   AIO_8B0E.RAW_NAME := 'Thermal Resistance - 3-wire (Cu10 climate - 426)';
   AIO_8B0E.___________0030_1 := false;
   AIO_8B0E.___________0030_2 := false;
   AIO_8B0E.PARAM_TYPE := 16#07;
   AIO_8B0E.PARAM_RANGE := 16#0E;
   AIO_8B0E.PARAM_COEF := 16#0B;
   AIO_8B0E.VALUE_COEF := 0.00426;
   AIO_8C0E.AIO_CODE := 16#8C0E;
   AIO_8C0E.___________0020_0 := false;
   AIO_8C0E.___________0010_2 := false;
   AIO_8C0E.RAW_MIN := -5000;
   AIO_8C0E.RAW_MAX := 15000;
   AIO_8C0E.RAW_NAME := 'Thermal Resistance - 3-wire (Cu10 climate - 427)';
   AIO_8C0E.___________0030_1 := false;
   AIO_8C0E.___________0030_2 := false;
   AIO_8C0E.PARAM_TYPE := 16#07;
   AIO_8C0E.PARAM_RANGE := 16#0E;
   AIO_8C0E.PARAM_COEF := 16#0C;
   AIO_8C0E.VALUE_COEF := 0.00427;
   AIO_8D0E.AIO_CODE := 16#8D0E;
   AIO_8D0E.___________0020_0 := false;
   AIO_8D0E.___________0010_2 := false;
   AIO_8D0E.RAW_MIN := -1800;
   AIO_8D0E.RAW_MAX := 15000;
   AIO_8D0E.RAW_NAME := 'Thermal Resistance - 3-wire (Cu10 climate - 428)';
   AIO_8D0E.___________0030_1 := false;
   AIO_8D0E.___________0030_2 := false;
   AIO_8D0E.PARAM_TYPE := 16#07;
   AIO_8D0E.PARAM_RANGE := 16#0E;
   AIO_8D0E.PARAM_COEF := 16#0D;
   AIO_8D0E.VALUE_COEF := 0.00428;
   AIO_8B0F.AIO_CODE := 16#8B0F;
   AIO_8B0F.___________0020_0 := false;
   AIO_8B0F.___________0010_2 := false;
   AIO_8B0F.RAW_MIN := -500;
   AIO_8B0F.RAW_MAX := 2000;
   AIO_8B0F.RAW_NAME := 'Thermal Resistance - 3-wire (Cu10 standard - 426)';
   AIO_8B0F.___________0030_1 := false;
   AIO_8B0F.___________0030_2 := false;
   AIO_8B0F.PARAM_TYPE := 16#07;
   AIO_8B0F.PARAM_RANGE := 16#0F;
   AIO_8B0F.PARAM_COEF := 16#0B;
   AIO_8B0F.VALUE_COEF := 0.00426;
   AIO_8C0F.AIO_CODE := 16#8C0F;
   AIO_8C0F.___________0020_0 := false;
   AIO_8C0F.___________0010_2 := false;
   AIO_8C0F.RAW_MIN := -2000;
   AIO_8C0F.RAW_MAX := 2600;
   AIO_8C0F.RAW_NAME := 'Thermal Resistance - 3-wire (Cu10 standard - 427)';
   AIO_8C0F.___________0030_1 := false;
   AIO_8C0F.___________0030_2 := false;
   AIO_8C0F.PARAM_TYPE := 16#07;
   AIO_8C0F.PARAM_RANGE := 16#0F;
   AIO_8C0F.PARAM_COEF := 16#0C;
   AIO_8C0F.VALUE_COEF := 0.00427;
   AIO_8D0F.AIO_CODE := 16#8D0F;
   AIO_8D0F.___________0020_0 := false;
   AIO_8D0F.___________0010_2 := false;
   AIO_8D0F.RAW_MIN := -1800;
   AIO_8D0F.RAW_MAX := 2000;
   AIO_8D0F.RAW_NAME := 'Thermal Resistance - 3-wire (Cu10 standard - 428)';
   AIO_8D0F.___________0030_1 := false;
   AIO_8D0F.___________0030_2 := false;
   AIO_8D0F.PARAM_TYPE := 16#07;
   AIO_8D0F.PARAM_RANGE := 16#0F;
   AIO_8D0F.PARAM_COEF := 16#0D;
   AIO_8D0F.VALUE_COEF := 0.00428;
   AIO_8B19.AIO_CODE := 16#8B19;
   AIO_8B19.___________0020_0 := false;
   AIO_8B19.___________0010_2 := false;
   AIO_8B19.RAW_MIN := -5000;
   AIO_8B19.RAW_MAX := 15000;
   AIO_8B19.RAW_NAME := 'Thermal Resistance - 3-wire (Cu50 climate - 426)';
   AIO_8B19.___________0030_1 := false;
   AIO_8B19.___________0030_2 := false;
   AIO_8B19.PARAM_TYPE := 16#07;
   AIO_8B19.PARAM_RANGE := 16#19;
   AIO_8B19.PARAM_COEF := 16#0B;
   AIO_8B19.VALUE_COEF := 0.00426;
   AIO_8C19.AIO_CODE := 16#8C19;
   AIO_8C19.___________0020_0 := false;
   AIO_8C19.___________0010_2 := false;
   AIO_8C19.RAW_MIN := -5000;
   AIO_8C19.RAW_MAX := 15000;
   AIO_8C19.RAW_NAME := 'Thermal Resistance - 3-wire (Cu50 climate - 427)';
   AIO_8C19.___________0030_1 := false;
   AIO_8C19.___________0030_2 := false;
   AIO_8C19.PARAM_TYPE := 16#07;
   AIO_8C19.PARAM_RANGE := 16#19;
   AIO_8C19.PARAM_COEF := 16#0C;
   AIO_8C19.VALUE_COEF := 0.00427;
   AIO_8D19.AIO_CODE := 16#8D19;
   AIO_8D19.___________0020_0 := false;
   AIO_8D19.___________0010_2 := false;
   AIO_8D19.RAW_MIN := -5000;
   AIO_8D19.RAW_MAX := 15000;
   AIO_8D19.RAW_NAME := 'Thermal Resistance - 3-wire (Cu50 climate - 428)';
   AIO_8D19.___________0030_1 := false;
   AIO_8D19.___________0030_2 := false;
   AIO_8D19.PARAM_TYPE := 16#07;
   AIO_8D19.PARAM_RANGE := 16#19;
   AIO_8D19.PARAM_COEF := 16#0D;
   AIO_8D19.VALUE_COEF := 0.00428;
   AIO_8B18.AIO_CODE := 16#8B18;
   AIO_8B18.___________0020_0 := false;
   AIO_8B18.___________0010_2 := false;
   AIO_8B18.RAW_MIN := -500;
   AIO_8B18.RAW_MAX := 2000;
   AIO_8B18.RAW_NAME := 'Thermal Resistance - 3-wire (Cu50 standard - 426)';
   AIO_8B18.___________0030_1 := false;
   AIO_8B18.___________0030_2 := false;
   AIO_8B18.PARAM_TYPE := 16#07;
   AIO_8B18.PARAM_RANGE := 16#18;
   AIO_8B18.PARAM_COEF := 16#0B;
   AIO_8B18.VALUE_COEF := 0.00426;
   AIO_8C18.AIO_CODE := 16#8C18;
   AIO_8C18.___________0020_0 := false;
   AIO_8C18.___________0010_2 := false;
   AIO_8C18.RAW_MIN := -2000;
   AIO_8C18.RAW_MAX := 2600;
   AIO_8C18.RAW_NAME := 'Thermal Resistance - 3-wire (Cu50 standard - 427)';
   AIO_8C18.___________0030_1 := false;
   AIO_8C18.___________0030_2 := false;
   AIO_8C18.PARAM_TYPE := 16#07;
   AIO_8C18.PARAM_RANGE := 16#18;
   AIO_8C18.PARAM_COEF := 16#0C;
   AIO_8C18.VALUE_COEF := 0.00427;
   AIO_8D18.AIO_CODE := 16#8D18;
   AIO_8D18.___________0020_0 := false;
   AIO_8D18.___________0010_2 := false;
   AIO_8D18.RAW_MIN := -1800;
   AIO_8D18.RAW_MAX := 2000;
   AIO_8D18.RAW_NAME := 'Thermal Resistance - 3-wire (Cu50 standard - 428)';
   AIO_8D18.___________0030_1 := false;
   AIO_8D18.___________0030_2 := false;
   AIO_8D18.PARAM_TYPE := 16#07;
   AIO_8D18.PARAM_RANGE := 16#18;
   AIO_8D18.PARAM_COEF := 16#0D;
   AIO_8D18.VALUE_COEF := 0.00428;
   AIO_8B1B.AIO_CODE := 16#8B1B;
   AIO_8B1B.___________0020_0 := false;
   AIO_8B1B.___________0010_2 := false;
   AIO_8B1B.RAW_MIN := -5000;
   AIO_8B1B.RAW_MAX := 15000;
   AIO_8B1B.RAW_NAME := 'Thermal Resistance - 3-wire (Cu100 climate - 426)';
   AIO_8B1B.___________0030_1 := false;
   AIO_8B1B.___________0030_2 := false;
   AIO_8B1B.PARAM_TYPE := 16#07;
   AIO_8B1B.PARAM_RANGE := 16#1B;
   AIO_8B1B.PARAM_COEF := 16#0B;
   AIO_8B1B.VALUE_COEF := 0.00426;
   AIO_8C1B.AIO_CODE := 16#8C1B;
   AIO_8C1B.___________0020_0 := false;
   AIO_8C1B.___________0010_2 := false;
   AIO_8C1B.RAW_MIN := -5000;
   AIO_8C1B.RAW_MAX := 15000;
   AIO_8C1B.RAW_NAME := 'Thermal Resistance - 3-wire (Cu100 climate - 427)';
   AIO_8C1B.___________0030_1 := false;
   AIO_8C1B.___________0030_2 := false;
   AIO_8C1B.PARAM_TYPE := 16#07;
   AIO_8C1B.PARAM_RANGE := 16#1B;
   AIO_8C1B.PARAM_COEF := 16#0C;
   AIO_8C1B.VALUE_COEF := 0.00427;
   AIO_8D1B.AIO_CODE := 16#8D1B;
   AIO_8D1B.___________0020_0 := false;
   AIO_8D1B.___________0010_2 := false;
   AIO_8D1B.RAW_MIN := -5000;
   AIO_8D1B.RAW_MAX := 15000;
   AIO_8D1B.RAW_NAME := 'Thermal Resistance - 3-wire (Cu100 climate - 428)';
   AIO_8D1B.___________0030_1 := false;
   AIO_8D1B.___________0030_2 := false;
   AIO_8D1B.PARAM_TYPE := 16#07;
   AIO_8D1B.PARAM_RANGE := 16#1B;
   AIO_8D1B.PARAM_COEF := 16#0D;
   AIO_8D1B.VALUE_COEF := 0.00428;
   AIO_8B1A.AIO_CODE := 16#8B1A;
   AIO_8B1A.___________0020_0 := false;
   AIO_8B1A.___________0010_2 := false;
   AIO_8B1A.RAW_MIN := -500;
   AIO_8B1A.RAW_MAX := 2000;
   AIO_8B1A.RAW_NAME := 'Thermal Resistance - 3-wire (Cu100 standard - 426)';
   AIO_8B1A.___________0030_1 := false;
   AIO_8B1A.___________0030_2 := false;
   AIO_8B1A.PARAM_TYPE := 16#07;
   AIO_8B1A.PARAM_RANGE := 16#1A;
   AIO_8B1A.PARAM_COEF := 16#0B;
   AIO_8B1A.VALUE_COEF := 0.00426;
   AIO_8C1A.AIO_CODE := 16#8C1A;
   AIO_8C1A.___________0020_0 := false;
   AIO_8C1A.___________0010_2 := false;
   AIO_8C1A.RAW_MIN := -2000;
   AIO_8C1A.RAW_MAX := 2600;
   AIO_8C1A.RAW_NAME := 'Thermal Resistance - 3-wire (Cu100 standard - 427)';
   AIO_8C1A.___________0030_1 := false;
   AIO_8C1A.___________0030_2 := false;
   AIO_8C1A.PARAM_TYPE := 16#07;
   AIO_8C1A.PARAM_RANGE := 16#1A;
   AIO_8C1A.PARAM_COEF := 16#0C;
   AIO_8C1A.VALUE_COEF := 0.00427;
   AIO_8D1A.AIO_CODE := 16#8D1A;
   AIO_8D1A.___________0020_0 := false;
   AIO_8D1A.___________0010_2 := false;
   AIO_8D1A.RAW_MIN := -1800;
   AIO_8D1A.RAW_MAX := 2000;
   AIO_8D1A.RAW_NAME := 'Thermal Resistance - 3-wire (Cu100 standard - 428)';
   AIO_8D1A.___________0030_1 := false;
   AIO_8D1A.___________0030_2 := false;
   AIO_8D1A.PARAM_TYPE := 16#07;
   AIO_8D1A.PARAM_RANGE := 16#1A;
   AIO_8D1A.PARAM_COEF := 16#0D;
   AIO_8D1A.VALUE_COEF := 0.00428;
   AIO_8A1D.AIO_CODE := 16#8A1D;
   AIO_8A1D.___________0020_0 := false;
   AIO_8A1D.___________0010_2 := false;
   AIO_8A1D.RAW_MIN := -6000;
   AIO_8A1D.RAW_MAX := 13000;
   AIO_8A1D.RAW_NAME := 'Thermal Resistance - 3-wire (LG-Ni1000 climate - 500)';
   AIO_8A1D.___________0030_1 := false;
   AIO_8A1D.___________0030_2 := false;
   AIO_8A1D.PARAM_TYPE := 16#07;
   AIO_8A1D.PARAM_RANGE := 16#1D;
   AIO_8A1D.PARAM_COEF := 16#0A;
   AIO_8A1D.VALUE_COEF := 0.005;
   AIO_8A1C.AIO_CODE := 16#8A1C;
   AIO_8A1C.___________0020_0 := false;
   AIO_8A1C.___________0010_2 := false;
   AIO_8A1C.RAW_MIN := -600;
   AIO_8A1C.RAW_MAX := 2500;
   AIO_8A1C.RAW_NAME := 'Thermal Resistance - 3-wire (LG-Ni1000 standard - 500)';
   AIO_8A1C.___________0030_1 := false;
   AIO_8A1C.___________0030_2 := false;
   AIO_8A1C.PARAM_TYPE := 16#07;
   AIO_8A1C.PARAM_RANGE := 16#1C;
   AIO_8A1C.PARAM_COEF := 16#0A;
   AIO_8A1C.VALUE_COEF := 0.005;
   AIO_871F.AIO_CODE := 16#871F;
   AIO_871F.___________0020_0 := false;
   AIO_871F.___________0010_2 := false;
   AIO_871F.RAW_MIN := -6000;
   AIO_871F.RAW_MAX := 13000;
   AIO_871F.RAW_NAME := 'Thermal Resistance - 3-wire (Ni10 climate - 617)';
   AIO_871F.___________0030_1 := false;
   AIO_871F.___________0030_2 := false;
   AIO_871F.PARAM_TYPE := 16#07;
   AIO_871F.PARAM_RANGE := 16#1F;
   AIO_871F.PARAM_COEF := 16#07;
   AIO_871F.VALUE_COEF := 0.00617;
   AIO_881F.AIO_CODE := 16#881F;
   AIO_881F.___________0020_0 := false;
   AIO_881F.___________0010_2 := false;
   AIO_881F.RAW_MIN := -6000;
   AIO_881F.RAW_MAX := 13000;
   AIO_881F.RAW_NAME := 'Thermal Resistance - 3-wire (Ni10 climate - 618)';
   AIO_881F.___________0030_1 := false;
   AIO_881F.___________0030_2 := false;
   AIO_881F.PARAM_TYPE := 16#07;
   AIO_881F.PARAM_RANGE := 16#1F;
   AIO_881F.PARAM_COEF := 16#08;
   AIO_881F.VALUE_COEF := 0.00618;
   AIO_891F.AIO_CODE := 16#891F;
   AIO_891F.___________0020_0 := false;
   AIO_891F.___________0010_2 := false;
   AIO_891F.RAW_MIN := -6000;
   AIO_891F.RAW_MAX := 13000;
   AIO_891F.RAW_NAME := 'Thermal Resistance - 3-wire (Ni10 climate - 672)';
   AIO_891F.___________0030_1 := false;
   AIO_891F.___________0030_2 := false;
   AIO_891F.PARAM_TYPE := 16#07;
   AIO_891F.PARAM_RANGE := 16#1F;
   AIO_891F.PARAM_COEF := 16#09;
   AIO_891F.VALUE_COEF := 0.00672;
   AIO_871E.AIO_CODE := 16#871E;
   AIO_871E.___________0020_0 := false;
   AIO_871E.___________0010_2 := false;
   AIO_871E.RAW_MIN := -600;
   AIO_871E.RAW_MAX := 1800;
   AIO_871E.RAW_NAME := 'Thermal Resistance - 3-wire (Ni10 standard - 617)';
   AIO_871E.___________0030_1 := false;
   AIO_871E.___________0030_2 := false;
   AIO_871E.PARAM_TYPE := 16#07;
   AIO_871E.PARAM_RANGE := 16#1E;
   AIO_871E.PARAM_COEF := 16#07;
   AIO_871E.VALUE_COEF := 0.00617;
   AIO_881E.AIO_CODE := 16#881E;
   AIO_881E.___________0020_0 := false;
   AIO_881E.___________0010_2 := false;
   AIO_881E.RAW_MIN := -600;
   AIO_881E.RAW_MAX := 2500;
   AIO_881E.RAW_NAME := 'Thermal Resistance - 3-wire (Ni10 standard - 618)';
   AIO_881E.___________0030_1 := false;
   AIO_881E.___________0030_2 := false;
   AIO_881E.PARAM_TYPE := 16#07;
   AIO_881E.PARAM_RANGE := 16#1E;
   AIO_881E.PARAM_COEF := 16#08;
   AIO_881E.VALUE_COEF := 0.00618;
   AIO_891E.AIO_CODE := 16#891E;
   AIO_891E.___________0020_0 := false;
   AIO_891E.___________0010_2 := false;
   AIO_891E.RAW_MIN := -600;
   AIO_891E.RAW_MAX := 2500;
   AIO_891E.RAW_NAME := 'Thermal Resistance - 3-wire (Ni10 standard - 672)';
   AIO_891E.___________0030_1 := false;
   AIO_891E.___________0030_2 := false;
   AIO_891E.PARAM_TYPE := 16#07;
   AIO_891E.PARAM_RANGE := 16#1E;
   AIO_891E.PARAM_COEF := 16#09;
   AIO_891E.VALUE_COEF := 0.00672;
   AIO_870D.AIO_CODE := 16#870D;
   AIO_870D.___________0020_0 := false;
   AIO_870D.___________0010_2 := false;
   AIO_870D.RAW_MIN := -6000;
   AIO_870D.RAW_MAX := 13000;
   AIO_870D.RAW_NAME := 'Thermal Resistance - 3-wire (Ni120 climate - 617)';
   AIO_870D.___________0030_1 := false;
   AIO_870D.___________0030_2 := false;
   AIO_870D.PARAM_TYPE := 16#07;
   AIO_870D.PARAM_RANGE := 16#0D;
   AIO_870D.PARAM_COEF := 16#07;
   AIO_870D.VALUE_COEF := 0.00617;
   AIO_880D.AIO_CODE := 16#880D;
   AIO_880D.___________0020_0 := false;
   AIO_880D.___________0010_2 := false;
   AIO_880D.RAW_MIN := -6000;
   AIO_880D.RAW_MAX := 13000;
   AIO_880D.RAW_NAME := 'Thermal Resistance - 3-wire (Ni120 climate - 618)';
   AIO_880D.___________0030_1 := false;
   AIO_880D.___________0030_2 := false;
   AIO_880D.PARAM_TYPE := 16#07;
   AIO_880D.PARAM_RANGE := 16#0D;
   AIO_880D.PARAM_COEF := 16#08;
   AIO_880D.VALUE_COEF := 0.00618;
   AIO_890D.AIO_CODE := 16#890D;
   AIO_890D.___________0020_0 := false;
   AIO_890D.___________0010_2 := false;
   AIO_890D.RAW_MIN := -6000;
   AIO_890D.RAW_MAX := 13000;
   AIO_890D.RAW_NAME := 'Thermal Resistance - 3-wire (Ni120 climate - 672)';
   AIO_890D.___________0030_1 := false;
   AIO_890D.___________0030_2 := false;
   AIO_890D.PARAM_TYPE := 16#07;
   AIO_890D.PARAM_RANGE := 16#0D;
   AIO_890D.PARAM_COEF := 16#09;
   AIO_890D.VALUE_COEF := 0.00672;
   AIO_870C.AIO_CODE := 16#870C;
   AIO_870C.___________0020_0 := false;
   AIO_870C.___________0010_2 := false;
   AIO_870C.RAW_MIN := -600;
   AIO_870C.RAW_MAX := 1800;
   AIO_870C.RAW_NAME := 'Thermal Resistance - 3-wire (Ni120 standard - 617)';
   AIO_870C.___________0030_1 := false;
   AIO_870C.___________0030_2 := false;
   AIO_870C.PARAM_TYPE := 16#07;
   AIO_870C.PARAM_RANGE := 16#0C;
   AIO_870C.PARAM_COEF := 16#07;
   AIO_870C.VALUE_COEF := 0.00617;
   AIO_880C.AIO_CODE := 16#880C;
   AIO_880C.___________0020_0 := false;
   AIO_880C.___________0010_2 := false;
   AIO_880C.RAW_MIN := -600;
   AIO_880C.RAW_MAX := 2500;
   AIO_880C.RAW_NAME := 'Thermal Resistance - 3-wire (Ni120 standard - 618)';
   AIO_880C.___________0030_1 := false;
   AIO_880C.___________0030_2 := false;
   AIO_880C.PARAM_TYPE := 16#07;
   AIO_880C.PARAM_RANGE := 16#0C;
   AIO_880C.PARAM_COEF := 16#08;
   AIO_880C.VALUE_COEF := 0.00618;
   AIO_890C.AIO_CODE := 16#890C;
   AIO_890C.___________0020_0 := false;
   AIO_890C.___________0010_2 := false;
   AIO_890C.RAW_MIN := -600;
   AIO_890C.RAW_MAX := 2500;
   AIO_890C.RAW_NAME := 'Thermal Resistance - 3-wire (Ni120 standard - 672)';
   AIO_890C.___________0030_1 := false;
   AIO_890C.___________0030_2 := false;
   AIO_890C.PARAM_TYPE := 16#07;
   AIO_890C.PARAM_RANGE := 16#0C;
   AIO_890C.PARAM_COEF := 16#09;
   AIO_890C.VALUE_COEF := 0.00672;
   AIO_8701.AIO_CODE := 16#8701;
   AIO_8701.___________0020_0 := false;
   AIO_8701.___________0010_2 := false;
   AIO_8701.RAW_MIN := -6000;
   AIO_8701.RAW_MAX := 13000;
   AIO_8701.RAW_NAME := 'Thermal Resistance - 3-wire (Ni100 climate - 617)';
   AIO_8701.___________0030_1 := false;
   AIO_8701.___________0030_2 := false;
   AIO_8701.PARAM_TYPE := 16#07;
   AIO_8701.PARAM_RANGE := 16#01;
   AIO_8701.PARAM_COEF := 16#07;
   AIO_8701.VALUE_COEF := 0.00617;
   AIO_8801.AIO_CODE := 16#8801;
   AIO_8801.___________0020_0 := false;
   AIO_8801.___________0010_2 := false;
   AIO_8801.RAW_MIN := -6000;
   AIO_8801.RAW_MAX := 13000;
   AIO_8801.RAW_NAME := 'Thermal Resistance - 3-wire (Ni100 climate - 618)';
   AIO_8801.___________0030_1 := false;
   AIO_8801.___________0030_2 := false;
   AIO_8801.PARAM_TYPE := 16#07;
   AIO_8801.PARAM_RANGE := 16#01;
   AIO_8801.PARAM_COEF := 16#08;
   AIO_8801.VALUE_COEF := 0.00618;
   AIO_8901.AIO_CODE := 16#8901;
   AIO_8901.___________0020_0 := false;
   AIO_8901.___________0010_2 := false;
   AIO_8901.RAW_MIN := -6000;
   AIO_8901.RAW_MAX := 13000;
   AIO_8901.RAW_NAME := 'Thermal Resistance - 3-wire (Ni100 climate - 672)';
   AIO_8901.___________0030_1 := false;
   AIO_8901.___________0030_2 := false;
   AIO_8901.PARAM_TYPE := 16#07;
   AIO_8901.PARAM_RANGE := 16#01;
   AIO_8901.PARAM_COEF := 16#09;
   AIO_8901.VALUE_COEF := 0.00672;
   AIO_8703.AIO_CODE := 16#8703;
   AIO_8703.___________0020_0 := false;
   AIO_8703.___________0010_2 := false;
   AIO_8703.RAW_MIN := -600;
   AIO_8703.RAW_MAX := 1800;
   AIO_8703.RAW_NAME := 'Thermal Resistance - 3-wire (Ni100 standard - 617)';
   AIO_8703.___________0030_1 := false;
   AIO_8703.___________0030_2 := false;
   AIO_8703.PARAM_TYPE := 16#07;
   AIO_8703.PARAM_RANGE := 16#03;
   AIO_8703.PARAM_COEF := 16#07;
   AIO_8703.VALUE_COEF := 0.00617;
   AIO_8803.AIO_CODE := 16#8803;
   AIO_8803.___________0020_0 := false;
   AIO_8803.___________0010_2 := false;
   AIO_8803.RAW_MIN := -600;
   AIO_8803.RAW_MAX := 2500;
   AIO_8803.RAW_NAME := 'Thermal Resistance - 3-wire (Ni100 standard - 618)';
   AIO_8803.___________0030_1 := false;
   AIO_8803.___________0030_2 := false;
   AIO_8803.PARAM_TYPE := 16#07;
   AIO_8803.PARAM_RANGE := 16#03;
   AIO_8803.PARAM_COEF := 16#08;
   AIO_8803.VALUE_COEF := 0.00618;
   AIO_8903.AIO_CODE := 16#8903;
   AIO_8903.___________0020_0 := false;
   AIO_8903.___________0010_2 := false;
   AIO_8903.RAW_MIN := -600;
   AIO_8903.RAW_MAX := 2500;
   AIO_8903.RAW_NAME := 'Thermal Resistance - 3-wire (Ni100 standard - 672)';
   AIO_8903.___________0030_1 := false;
   AIO_8903.___________0030_2 := false;
   AIO_8903.PARAM_TYPE := 16#07;
   AIO_8903.PARAM_RANGE := 16#03;
   AIO_8903.PARAM_COEF := 16#09;
   AIO_8903.VALUE_COEF := 0.00672;
   AIO_8711.AIO_CODE := 16#8711;
   AIO_8711.___________0020_0 := false;
   AIO_8711.___________0010_2 := false;
   AIO_8711.RAW_MIN := -6000;
   AIO_8711.RAW_MAX := 13000;
   AIO_8711.RAW_NAME := 'Thermal Resistance - 3-wire (Ni200 climate - 617)';
   AIO_8711.___________0030_1 := false;
   AIO_8711.___________0030_2 := false;
   AIO_8711.PARAM_TYPE := 16#07;
   AIO_8711.PARAM_RANGE := 16#11;
   AIO_8711.PARAM_COEF := 16#07;
   AIO_8711.VALUE_COEF := 0.00617;
   AIO_8811.AIO_CODE := 16#8811;
   AIO_8811.___________0020_0 := false;
   AIO_8811.___________0010_2 := false;
   AIO_8811.RAW_MIN := -6000;
   AIO_8811.RAW_MAX := 13000;
   AIO_8811.RAW_NAME := 'Thermal Resistance - 3-wire (Ni200 climate - 618)';
   AIO_8811.___________0030_1 := false;
   AIO_8811.___________0030_2 := false;
   AIO_8811.PARAM_TYPE := 16#07;
   AIO_8811.PARAM_RANGE := 16#11;
   AIO_8811.PARAM_COEF := 16#08;
   AIO_8811.VALUE_COEF := 0.00618;
   AIO_8911.AIO_CODE := 16#8911;
   AIO_8911.___________0020_0 := false;
   AIO_8911.___________0010_2 := false;
   AIO_8911.RAW_MIN := -6000;
   AIO_8911.RAW_MAX := 13000;
   AIO_8911.RAW_NAME := 'Thermal Resistance - 3-wire (Ni200 climate - 672)';
   AIO_8911.___________0030_1 := false;
   AIO_8911.___________0030_2 := false;
   AIO_8911.PARAM_TYPE := 16#07;
   AIO_8911.PARAM_RANGE := 16#11;
   AIO_8911.PARAM_COEF := 16#09;
   AIO_8911.VALUE_COEF := 0.00672;
   AIO_8710.AIO_CODE := 16#8710;
   AIO_8710.___________0020_0 := false;
   AIO_8710.___________0010_2 := false;
   AIO_8710.RAW_MIN := -600;
   AIO_8710.RAW_MAX := 1800;
   AIO_8710.RAW_NAME := 'Thermal Resistance - 3-wire (Ni200 standard - 617)';
   AIO_8710.___________0030_1 := false;
   AIO_8710.___________0030_2 := false;
   AIO_8710.PARAM_TYPE := 16#07;
   AIO_8710.PARAM_RANGE := 16#10;
   AIO_8710.PARAM_COEF := 16#07;
   AIO_8710.VALUE_COEF := 0.00617;
   AIO_8810.AIO_CODE := 16#8810;
   AIO_8810.___________0020_0 := false;
   AIO_8810.___________0010_2 := false;
   AIO_8810.RAW_MIN := -600;
   AIO_8810.RAW_MAX := 2500;
   AIO_8810.RAW_NAME := 'Thermal Resistance - 3-wire (Ni200 standard - 618)';
   AIO_8810.___________0030_1 := false;
   AIO_8810.___________0030_2 := false;
   AIO_8810.PARAM_TYPE := 16#07;
   AIO_8810.PARAM_RANGE := 16#10;
   AIO_8810.PARAM_COEF := 16#08;
   AIO_8810.VALUE_COEF := 0.00618;
   AIO_8910.AIO_CODE := 16#8910;
   AIO_8910.___________0020_0 := false;
   AIO_8910.___________0010_2 := false;
   AIO_8910.RAW_MIN := -600;
   AIO_8910.RAW_MAX := 2500;
   AIO_8910.RAW_NAME := 'Thermal Resistance - 3-wire (Ni200 standard - 672)';
   AIO_8910.___________0030_1 := false;
   AIO_8910.___________0030_2 := false;
   AIO_8910.PARAM_TYPE := 16#07;
   AIO_8910.PARAM_RANGE := 16#10;
   AIO_8910.PARAM_COEF := 16#09;
   AIO_8910.VALUE_COEF := 0.00672;
   AIO_8713.AIO_CODE := 16#8713;
   AIO_8713.___________0020_0 := false;
   AIO_8713.___________0010_2 := false;
   AIO_8713.RAW_MIN := -6000;
   AIO_8713.RAW_MAX := 13000;
   AIO_8713.RAW_NAME := 'Thermal Resistance - 3-wire (Ni500 climate - 617)';
   AIO_8713.___________0030_1 := false;
   AIO_8713.___________0030_2 := false;
   AIO_8713.PARAM_TYPE := 16#07;
   AIO_8713.PARAM_RANGE := 16#13;
   AIO_8713.PARAM_COEF := 16#07;
   AIO_8713.VALUE_COEF := 0.00617;
   AIO_8813.AIO_CODE := 16#8813;
   AIO_8813.___________0020_0 := false;
   AIO_8813.___________0010_2 := false;
   AIO_8813.RAW_MIN := -6000;
   AIO_8813.RAW_MAX := 13000;
   AIO_8813.RAW_NAME := 'Thermal Resistance - 3-wire (Ni500 climate - 618)';
   AIO_8813.___________0030_1 := false;
   AIO_8813.___________0030_2 := false;
   AIO_8813.PARAM_TYPE := 16#07;
   AIO_8813.PARAM_RANGE := 16#13;
   AIO_8813.PARAM_COEF := 16#08;
   AIO_8813.VALUE_COEF := 0.00618;
   AIO_8913.AIO_CODE := 16#8913;
   AIO_8913.___________0020_0 := false;
   AIO_8913.___________0010_2 := false;
   AIO_8913.RAW_MIN := -6000;
   AIO_8913.RAW_MAX := 13000;
   AIO_8913.RAW_NAME := 'Thermal Resistance - 3-wire (Ni500 climate - 672)';
   AIO_8913.___________0030_1 := false;
   AIO_8913.___________0030_2 := false;
   AIO_8913.PARAM_TYPE := 16#07;
   AIO_8913.PARAM_RANGE := 16#13;
   AIO_8913.PARAM_COEF := 16#09;
   AIO_8913.VALUE_COEF := 0.00672;
   AIO_8712.AIO_CODE := 16#8712;
   AIO_8712.___________0020_0 := false;
   AIO_8712.___________0010_2 := false;
   AIO_8712.RAW_MIN := -600;
   AIO_8712.RAW_MAX := 1800;
   AIO_8712.RAW_NAME := 'Thermal Resistance - 3-wire (Ni500 standard - 617)';
   AIO_8712.___________0030_1 := false;
   AIO_8712.___________0030_2 := false;
   AIO_8712.PARAM_TYPE := 16#07;
   AIO_8712.PARAM_RANGE := 16#12;
   AIO_8712.PARAM_COEF := 16#07;
   AIO_8712.VALUE_COEF := 0.00617;
   AIO_8812.AIO_CODE := 16#8812;
   AIO_8812.___________0020_0 := false;
   AIO_8812.___________0010_2 := false;
   AIO_8812.RAW_MIN := -600;
   AIO_8812.RAW_MAX := 2500;
   AIO_8812.RAW_NAME := 'Thermal Resistance - 3-wire (Ni500 standard - 618)';
   AIO_8812.___________0030_1 := false;
   AIO_8812.___________0030_2 := false;
   AIO_8812.PARAM_TYPE := 16#07;
   AIO_8812.PARAM_RANGE := 16#12;
   AIO_8812.PARAM_COEF := 16#08;
   AIO_8812.VALUE_COEF := 0.00618;
   AIO_8912.AIO_CODE := 16#8912;
   AIO_8912.___________0020_0 := false;
   AIO_8912.___________0010_2 := false;
   AIO_8912.RAW_MIN := -600;
   AIO_8912.RAW_MAX := 2500;
   AIO_8912.RAW_NAME := 'Thermal Resistance - 3-wire (Ni500 standard - 672)';
   AIO_8912.___________0030_1 := false;
   AIO_8912.___________0030_2 := false;
   AIO_8912.PARAM_TYPE := 16#07;
   AIO_8912.PARAM_RANGE := 16#12;
   AIO_8912.PARAM_COEF := 16#09;
   AIO_8912.VALUE_COEF := 0.00672;
   AIO_870A.AIO_CODE := 16#870A;
   AIO_870A.___________0020_0 := false;
   AIO_870A.___________0010_2 := false;
   AIO_870A.RAW_MIN := -6000;
   AIO_870A.RAW_MAX := 13000;
   AIO_870A.RAW_NAME := 'Thermal Resistance - 3-wire (Ni1000 climate - 617)';
   AIO_870A.___________0030_1 := false;
   AIO_870A.___________0030_2 := false;
   AIO_870A.PARAM_TYPE := 16#07;
   AIO_870A.PARAM_RANGE := 16#0A;
   AIO_870A.PARAM_COEF := 16#07;
   AIO_870A.VALUE_COEF := 0.00617;
   AIO_880A.AIO_CODE := 16#880A;
   AIO_880A.___________0020_0 := false;
   AIO_880A.___________0010_2 := false;
   AIO_880A.RAW_MIN := -6000;
   AIO_880A.RAW_MAX := 13000;
   AIO_880A.RAW_NAME := 'Thermal Resistance - 3-wire (Ni1000 climate - 618)';
   AIO_880A.___________0030_1 := false;
   AIO_880A.___________0030_2 := false;
   AIO_880A.PARAM_TYPE := 16#07;
   AIO_880A.PARAM_RANGE := 16#0A;
   AIO_880A.PARAM_COEF := 16#08;
   AIO_880A.VALUE_COEF := 0.00618;
   AIO_890A.AIO_CODE := 16#890A;
   AIO_890A.___________0020_0 := false;
   AIO_890A.___________0010_2 := false;
   AIO_890A.RAW_MIN := -6000;
   AIO_890A.RAW_MAX := 13000;
   AIO_890A.RAW_NAME := 'Thermal Resistance - 3-wire (Ni1000 climate - 672)';
   AIO_890A.___________0030_1 := false;
   AIO_890A.___________0030_2 := false;
   AIO_890A.PARAM_TYPE := 16#07;
   AIO_890A.PARAM_RANGE := 16#0A;
   AIO_890A.PARAM_COEF := 16#09;
   AIO_890A.VALUE_COEF := 0.00672;
   AIO_8706.AIO_CODE := 16#8706;
   AIO_8706.___________0020_0 := false;
   AIO_8706.___________0010_2 := false;
   AIO_8706.RAW_MIN := -600;
   AIO_8706.RAW_MAX := 1800;
   AIO_8706.RAW_NAME := 'Thermal Resistance - 3-wire (Ni1000 standard - 617)';
   AIO_8706.___________0030_1 := false;
   AIO_8706.___________0030_2 := false;
   AIO_8706.PARAM_TYPE := 16#07;
   AIO_8706.PARAM_RANGE := 16#06;
   AIO_8706.PARAM_COEF := 16#07;
   AIO_8706.VALUE_COEF := 0.00617;
   AIO_8806.AIO_CODE := 16#8806;
   AIO_8806.___________0020_0 := false;
   AIO_8806.___________0010_2 := false;
   AIO_8806.RAW_MIN := -600;
   AIO_8806.RAW_MAX := 2500;
   AIO_8806.RAW_NAME := 'Thermal Resistance - 3-wire (Ni1000 standard - 618)';
   AIO_8806.___________0030_1 := false;
   AIO_8806.___________0030_2 := false;
   AIO_8806.PARAM_TYPE := 16#07;
   AIO_8806.PARAM_RANGE := 16#06;
   AIO_8806.PARAM_COEF := 16#08;
   AIO_8806.VALUE_COEF := 0.00618;
   AIO_8906.AIO_CODE := 16#8906;
   AIO_8906.___________0020_0 := false;
   AIO_8906.___________0010_2 := false;
   AIO_8906.RAW_MIN := -600;
   AIO_8906.RAW_MAX := 2500;
   AIO_8906.RAW_NAME := 'Thermal Resistance - 3-wire (Ni1000 standard - 672)';
   AIO_8906.___________0030_1 := false;
   AIO_8906.___________0030_2 := false;
   AIO_8906.PARAM_TYPE := 16#07;
   AIO_8906.PARAM_RANGE := 16#06;
   AIO_8906.PARAM_COEF := 16#09;
   AIO_8906.VALUE_COEF := 0.00672;
   AIO_8015.AIO_CODE := 16#8015;
   AIO_8015.___________0020_0 := false;
   AIO_8015.___________0010_2 := false;
   AIO_8015.RAW_MIN := -12000;
   AIO_8015.RAW_MAX := 13000;
   AIO_8015.RAW_NAME := 'Thermal Resistance - 3-wire (Pt10 climate - 3851)';
   AIO_8015.___________0030_1 := false;
   AIO_8015.___________0030_2 := false;
   AIO_8015.PARAM_TYPE := 16#07;
   AIO_8015.PARAM_RANGE := 16#15;
   AIO_8015.PARAM_COEF := 16#00;
   AIO_8015.VALUE_COEF := 0.003851;
   AIO_8215.AIO_CODE := 16#8215;
   AIO_8215.___________0020_0 := false;
   AIO_8215.___________0010_2 := false;
   AIO_8215.RAW_MIN := -12000;
   AIO_8215.RAW_MAX := 13000;
   AIO_8215.RAW_NAME := 'Thermal Resistance - 3-wire (Pt10 climate - 3902)';
   AIO_8215.___________0030_1 := false;
   AIO_8215.___________0030_2 := false;
   AIO_8215.PARAM_TYPE := 16#07;
   AIO_8215.PARAM_RANGE := 16#15;
   AIO_8215.PARAM_COEF := 16#02;
   AIO_8215.VALUE_COEF := 0.003902;
   AIO_8515.AIO_CODE := 16#8515;
   AIO_8515.___________0020_0 := false;
   AIO_8515.___________0010_2 := false;
   AIO_8515.RAW_MIN := -12000;
   AIO_8515.RAW_MAX := 13000;
   AIO_8515.RAW_NAME := 'Thermal Resistance - 3-wire (Pt10 climate - 391)';
   AIO_8515.___________0030_1 := false;
   AIO_8515.___________0030_2 := false;
   AIO_8515.PARAM_TYPE := 16#07;
   AIO_8515.PARAM_RANGE := 16#15;
   AIO_8515.PARAM_COEF := 16#05;
   AIO_8515.VALUE_COEF := 0.00391;
   AIO_8115.AIO_CODE := 16#8115;
   AIO_8115.___________0020_0 := false;
   AIO_8115.___________0010_2 := false;
   AIO_8115.RAW_MIN := -12000;
   AIO_8115.RAW_MAX := 13000;
   AIO_8115.RAW_NAME := 'Thermal Resistance - 3-wire (Pt10 climate - 3916)';
   AIO_8115.___________0030_1 := false;
   AIO_8115.___________0030_2 := false;
   AIO_8115.PARAM_TYPE := 16#07;
   AIO_8115.PARAM_RANGE := 16#15;
   AIO_8115.PARAM_COEF := 16#01;
   AIO_8115.VALUE_COEF := 0.003916;
   AIO_8315.AIO_CODE := 16#8315;
   AIO_8315.___________0020_0 := false;
   AIO_8315.___________0010_2 := false;
   AIO_8315.RAW_MIN := -12000;
   AIO_8315.RAW_MAX := 13000;
   AIO_8315.RAW_NAME := 'Thermal Resistance - 3-wire (Pt10 climate - 392)';
   AIO_8315.___________0030_1 := false;
   AIO_8315.___________0030_2 := false;
   AIO_8315.PARAM_TYPE := 16#07;
   AIO_8315.PARAM_RANGE := 16#15;
   AIO_8315.PARAM_COEF := 16#03;
   AIO_8315.VALUE_COEF := 0.00392;
   AIO_8014.AIO_CODE := 16#8014;
   AIO_8014.___________0020_0 := false;
   AIO_8014.___________0010_2 := false;
   AIO_8014.RAW_MIN := -2000;
   AIO_8014.RAW_MAX := 8500;
   AIO_8014.RAW_NAME := 'Thermal Resistance - 3-wire (Pt10 standard - 3851)';
   AIO_8014.___________0030_1 := false;
   AIO_8014.___________0030_2 := false;
   AIO_8014.PARAM_TYPE := 16#07;
   AIO_8014.PARAM_RANGE := 16#14;
   AIO_8014.PARAM_COEF := 16#00;
   AIO_8014.VALUE_COEF := 0.003851;
   AIO_8214.AIO_CODE := 16#8214;
   AIO_8214.___________0020_0 := false;
   AIO_8214.___________0010_2 := false;
   AIO_8214.RAW_MIN := -2000;
   AIO_8214.RAW_MAX := 8500;
   AIO_8214.RAW_NAME := 'Thermal Resistance - 3-wire (Pt10 standard - 3902)';
   AIO_8214.___________0030_1 := false;
   AIO_8214.___________0030_2 := false;
   AIO_8214.PARAM_TYPE := 16#07;
   AIO_8214.PARAM_RANGE := 16#14;
   AIO_8214.PARAM_COEF := 16#02;
   AIO_8214.VALUE_COEF := 0.003902;
   AIO_8514.AIO_CODE := 16#8514;
   AIO_8514.___________0020_0 := false;
   AIO_8514.___________0010_2 := false;
   AIO_8514.RAW_MIN := -2000;
   AIO_8514.RAW_MAX := 8500;
   AIO_8514.RAW_NAME := 'Thermal Resistance - 3-wire (Pt10 standard - 391)';
   AIO_8514.___________0030_1 := false;
   AIO_8514.___________0030_2 := false;
   AIO_8514.PARAM_TYPE := 16#07;
   AIO_8514.PARAM_RANGE := 16#14;
   AIO_8514.PARAM_COEF := 16#05;
   AIO_8514.VALUE_COEF := 0.00391;
   AIO_8114.AIO_CODE := 16#8114;
   AIO_8114.___________0020_0 := false;
   AIO_8114.___________0010_2 := false;
   AIO_8114.RAW_MIN := -2000;
   AIO_8114.RAW_MAX := 8500;
   AIO_8114.RAW_NAME := 'Thermal Resistance - 3-wire (Pt10 standard - 3916)';
   AIO_8114.___________0030_1 := false;
   AIO_8114.___________0030_2 := false;
   AIO_8114.PARAM_TYPE := 16#07;
   AIO_8114.PARAM_RANGE := 16#14;
   AIO_8114.PARAM_COEF := 16#01;
   AIO_8114.VALUE_COEF := 0.003916;
   AIO_8314.AIO_CODE := 16#8314;
   AIO_8314.___________0020_0 := false;
   AIO_8314.___________0010_2 := false;
   AIO_8314.RAW_MIN := -2000;
   AIO_8314.RAW_MAX := 8500;
   AIO_8314.RAW_NAME := 'Thermal Resistance - 3-wire (Pt10 standard - 392)';
   AIO_8314.___________0030_1 := false;
   AIO_8314.___________0030_2 := false;
   AIO_8314.PARAM_TYPE := 16#07;
   AIO_8314.PARAM_RANGE := 16#14;
   AIO_8314.PARAM_COEF := 16#03;
   AIO_8314.VALUE_COEF := 0.00392;
   AIO_8017.AIO_CODE := 16#8017;
   AIO_8017.___________0020_0 := false;
   AIO_8017.___________0010_2 := false;
   AIO_8017.RAW_MIN := -12000;
   AIO_8017.RAW_MAX := 13000;
   AIO_8017.RAW_NAME := 'Thermal Resistance - 3-wire (Pt50 climate - 3851)';
   AIO_8017.___________0030_1 := false;
   AIO_8017.___________0030_2 := false;
   AIO_8017.PARAM_TYPE := 16#07;
   AIO_8017.PARAM_RANGE := 16#17;
   AIO_8017.PARAM_COEF := 16#00;
   AIO_8017.VALUE_COEF := 0.003851;
   AIO_8217.AIO_CODE := 16#8217;
   AIO_8217.___________0020_0 := false;
   AIO_8217.___________0010_2 := false;
   AIO_8217.RAW_MIN := -12000;
   AIO_8217.RAW_MAX := 13000;
   AIO_8217.RAW_NAME := 'Thermal Resistance - 3-wire (Pt50 climate - 3902)';
   AIO_8217.___________0030_1 := false;
   AIO_8217.___________0030_2 := false;
   AIO_8217.PARAM_TYPE := 16#07;
   AIO_8217.PARAM_RANGE := 16#17;
   AIO_8217.PARAM_COEF := 16#02;
   AIO_8217.VALUE_COEF := 0.003902;
   AIO_8517.AIO_CODE := 16#8517;
   AIO_8517.___________0020_0 := false;
   AIO_8517.___________0010_2 := false;
   AIO_8517.RAW_MIN := -12000;
   AIO_8517.RAW_MAX := 13000;
   AIO_8517.RAW_NAME := 'Thermal Resistance - 3-wire (Pt50 climate - 391)';
   AIO_8517.___________0030_1 := false;
   AIO_8517.___________0030_2 := false;
   AIO_8517.PARAM_TYPE := 16#07;
   AIO_8517.PARAM_RANGE := 16#17;
   AIO_8517.PARAM_COEF := 16#05;
   AIO_8517.VALUE_COEF := 0.00391;
   AIO_8117.AIO_CODE := 16#8117;
   AIO_8117.___________0020_0 := false;
   AIO_8117.___________0010_2 := false;
   AIO_8117.RAW_MIN := -12000;
   AIO_8117.RAW_MAX := 13000;
   AIO_8117.RAW_NAME := 'Thermal Resistance - 3-wire (Pt50 climate - 3916)';
   AIO_8117.___________0030_1 := false;
   AIO_8117.___________0030_2 := false;
   AIO_8117.PARAM_TYPE := 16#07;
   AIO_8117.PARAM_RANGE := 16#17;
   AIO_8117.PARAM_COEF := 16#01;
   AIO_8117.VALUE_COEF := 0.003916;
   AIO_8317.AIO_CODE := 16#8317;
   AIO_8317.___________0020_0 := false;
   AIO_8317.___________0010_2 := false;
   AIO_8317.RAW_MIN := -12000;
   AIO_8317.RAW_MAX := 13000;
   AIO_8317.RAW_NAME := 'Thermal Resistance - 3-wire (Pt50 climate - 392)';
   AIO_8317.___________0030_1 := false;
   AIO_8317.___________0030_2 := false;
   AIO_8317.PARAM_TYPE := 16#07;
   AIO_8317.PARAM_RANGE := 16#17;
   AIO_8317.PARAM_COEF := 16#03;
   AIO_8317.VALUE_COEF := 0.00392;
   AIO_8016.AIO_CODE := 16#8016;
   AIO_8016.___________0020_0 := false;
   AIO_8016.___________0010_2 := false;
   AIO_8016.RAW_MIN := -2000;
   AIO_8016.RAW_MAX := 8500;
   AIO_8016.RAW_NAME := 'Thermal Resistance - 3-wire (Pt50 standard - 3851)';
   AIO_8016.___________0030_1 := false;
   AIO_8016.___________0030_2 := false;
   AIO_8016.PARAM_TYPE := 16#07;
   AIO_8016.PARAM_RANGE := 16#16;
   AIO_8016.PARAM_COEF := 16#00;
   AIO_8016.VALUE_COEF := 0.003851;
   AIO_8216.AIO_CODE := 16#8216;
   AIO_8216.___________0020_0 := false;
   AIO_8216.___________0010_2 := false;
   AIO_8216.RAW_MIN := -2000;
   AIO_8216.RAW_MAX := 8500;
   AIO_8216.RAW_NAME := 'Thermal Resistance - 3-wire (Pt50 standard - 3902)';
   AIO_8216.___________0030_1 := false;
   AIO_8216.___________0030_2 := false;
   AIO_8216.PARAM_TYPE := 16#07;
   AIO_8216.PARAM_RANGE := 16#16;
   AIO_8216.PARAM_COEF := 16#02;
   AIO_8216.VALUE_COEF := 0.003902;
   AIO_8516.AIO_CODE := 16#8516;
   AIO_8516.___________0020_0 := false;
   AIO_8516.___________0010_2 := false;
   AIO_8516.RAW_MIN := -2000;
   AIO_8516.RAW_MAX := 8500;
   AIO_8516.RAW_NAME := 'Thermal Resistance - 3-wire (Pt50 standard - 391)';
   AIO_8516.___________0030_1 := false;
   AIO_8516.___________0030_2 := false;
   AIO_8516.PARAM_TYPE := 16#07;
   AIO_8516.PARAM_RANGE := 16#16;
   AIO_8516.PARAM_COEF := 16#05;
   AIO_8516.VALUE_COEF := 0.00391;
   AIO_8116.AIO_CODE := 16#8116;
   AIO_8116.___________0020_0 := false;
   AIO_8116.___________0010_2 := false;
   AIO_8116.RAW_MIN := -2000;
   AIO_8116.RAW_MAX := 8500;
   AIO_8116.RAW_NAME := 'Thermal Resistance - 3-wire (Pt50 standard - 3916)';
   AIO_8116.___________0030_1 := false;
   AIO_8116.___________0030_2 := false;
   AIO_8116.PARAM_TYPE := 16#07;
   AIO_8116.PARAM_RANGE := 16#16;
   AIO_8116.PARAM_COEF := 16#01;
   AIO_8116.VALUE_COEF := 0.003916;
   AIO_8316.AIO_CODE := 16#8316;
   AIO_8316.___________0020_0 := false;
   AIO_8316.___________0010_2 := false;
   AIO_8316.RAW_MIN := -2000;
   AIO_8316.RAW_MAX := 8500;
   AIO_8316.RAW_NAME := 'Thermal Resistance - 3-wire (Pt50 standard - 392)';
   AIO_8316.___________0030_1 := false;
   AIO_8316.___________0030_2 := false;
   AIO_8316.PARAM_TYPE := 16#07;
   AIO_8316.PARAM_RANGE := 16#16;
   AIO_8316.PARAM_COEF := 16#03;
   AIO_8316.VALUE_COEF := 0.00392;
   AIO_8000.AIO_CODE := 16#8000;
   AIO_8000.___________0020_0 := false;
   AIO_8000.___________0010_2 := false;
   AIO_8000.RAW_MIN := -12000;
   AIO_8000.RAW_MAX := 13000;
   AIO_8000.RAW_NAME := 'Thermal Resistance - 3-wire (Pt100 climate - 3851)';
   AIO_8000.___________0030_1 := false;
   AIO_8000.___________0030_2 := false;
   AIO_8000.PARAM_TYPE := 16#07;
   AIO_8000.PARAM_RANGE := 16#00;
   AIO_8000.PARAM_COEF := 16#00;
   AIO_8000.VALUE_COEF := 0.003851;
   AIO_8200.AIO_CODE := 16#8200;
   AIO_8200.___________0020_0 := false;
   AIO_8200.___________0010_2 := false;
   AIO_8200.RAW_MIN := -12000;
   AIO_8200.RAW_MAX := 13000;
   AIO_8200.RAW_NAME := 'Thermal Resistance - 3-wire (Pt100 climate - 3902)';
   AIO_8200.___________0030_1 := false;
   AIO_8200.___________0030_2 := false;
   AIO_8200.PARAM_TYPE := 16#07;
   AIO_8200.PARAM_RANGE := 16#00;
   AIO_8200.PARAM_COEF := 16#02;
   AIO_8200.VALUE_COEF := 0.003902;
   AIO_8500.AIO_CODE := 16#8500;
   AIO_8500.___________0020_0 := false;
   AIO_8500.___________0010_2 := false;
   AIO_8500.RAW_MIN := -12000;
   AIO_8500.RAW_MAX := 13000;
   AIO_8500.RAW_NAME := 'Thermal Resistance - 3-wire (Pt100 climate - 391)';
   AIO_8500.___________0030_1 := false;
   AIO_8500.___________0030_2 := false;
   AIO_8500.PARAM_TYPE := 16#07;
   AIO_8500.PARAM_RANGE := 16#00;
   AIO_8500.PARAM_COEF := 16#05;
   AIO_8500.VALUE_COEF := 0.00391;
   AIO_8100.AIO_CODE := 16#8100;
   AIO_8100.___________0020_0 := false;
   AIO_8100.___________0010_2 := false;
   AIO_8100.RAW_MIN := -12000;
   AIO_8100.RAW_MAX := 13000;
   AIO_8100.RAW_NAME := 'Thermal Resistance - 3-wire (Pt100 climate - 3916)';
   AIO_8100.___________0030_1 := false;
   AIO_8100.___________0030_2 := false;
   AIO_8100.PARAM_TYPE := 16#07;
   AIO_8100.PARAM_RANGE := 16#00;
   AIO_8100.PARAM_COEF := 16#01;
   AIO_8100.VALUE_COEF := 0.003916;
   AIO_8300.AIO_CODE := 16#8300;
   AIO_8300.___________0020_0 := false;
   AIO_8300.___________0010_2 := false;
   AIO_8300.RAW_MIN := -12000;
   AIO_8300.RAW_MAX := 13000;
   AIO_8300.RAW_NAME := 'Thermal Resistance - 3-wire (Pt100 climate - 392)';
   AIO_8300.___________0030_1 := false;
   AIO_8300.___________0030_2 := false;
   AIO_8300.PARAM_TYPE := 16#07;
   AIO_8300.PARAM_RANGE := 16#00;
   AIO_8300.PARAM_COEF := 16#03;
   AIO_8300.VALUE_COEF := 0.00392;
   AIO_8002.AIO_CODE := 16#8002;
   AIO_8002.___________0020_0 := false;
   AIO_8002.___________0010_2 := false;
   AIO_8002.RAW_MIN := -2000;
   AIO_8002.RAW_MAX := 8500;
   AIO_8002.RAW_NAME := 'Thermal Resistance - 3-wire (Pt100 standard - 3851)';
   AIO_8002.___________0030_1 := false;
   AIO_8002.___________0030_2 := false;
   AIO_8002.PARAM_TYPE := 16#07;
   AIO_8002.PARAM_RANGE := 16#02;
   AIO_8002.PARAM_COEF := 16#00;
   AIO_8002.VALUE_COEF := 0.003851;
   AIO_8202.AIO_CODE := 16#8202;
   AIO_8202.___________0020_0 := false;
   AIO_8202.___________0010_2 := false;
   AIO_8202.RAW_MIN := -2000;
   AIO_8202.RAW_MAX := 8500;
   AIO_8202.RAW_NAME := 'Thermal Resistance - 3-wire (Pt100 standard - 3902)';
   AIO_8202.___________0030_1 := false;
   AIO_8202.___________0030_2 := false;
   AIO_8202.PARAM_TYPE := 16#07;
   AIO_8202.PARAM_RANGE := 16#02;
   AIO_8202.PARAM_COEF := 16#02;
   AIO_8202.VALUE_COEF := 0.003902;
   AIO_8502.AIO_CODE := 16#8502;
   AIO_8502.___________0020_0 := false;
   AIO_8502.___________0010_2 := false;
   AIO_8502.RAW_MIN := -2000;
   AIO_8502.RAW_MAX := 8500;
   AIO_8502.RAW_NAME := 'Thermal Resistance - 3-wire (Pt100 standard - 391)';
   AIO_8502.___________0030_1 := false;
   AIO_8502.___________0030_2 := false;
   AIO_8502.PARAM_TYPE := 16#07;
   AIO_8502.PARAM_RANGE := 16#02;
   AIO_8502.PARAM_COEF := 16#05;
   AIO_8502.VALUE_COEF := 0.00391;
   AIO_8102.AIO_CODE := 16#8102;
   AIO_8102.___________0020_0 := false;
   AIO_8102.___________0010_2 := false;
   AIO_8102.RAW_MIN := -2000;
   AIO_8102.RAW_MAX := 8500;
   AIO_8102.RAW_NAME := 'Thermal Resistance - 3-wire (Pt100 standard - 3916)';
   AIO_8102.___________0030_1 := false;
   AIO_8102.___________0030_2 := false;
   AIO_8102.PARAM_TYPE := 16#07;
   AIO_8102.PARAM_RANGE := 16#02;
   AIO_8102.PARAM_COEF := 16#01;
   AIO_8102.VALUE_COEF := 0.003916;
   AIO_8302.AIO_CODE := 16#8302;
   AIO_8302.___________0020_0 := false;
   AIO_8302.___________0010_2 := false;
   AIO_8302.RAW_MIN := -2000;
   AIO_8302.RAW_MAX := 8500;
   AIO_8302.RAW_NAME := 'Thermal Resistance - 3-wire (Pt100 standard - 392)';
   AIO_8302.___________0030_1 := false;
   AIO_8302.___________0030_2 := false;
   AIO_8302.PARAM_TYPE := 16#07;
   AIO_8302.PARAM_RANGE := 16#02;
   AIO_8302.PARAM_COEF := 16#03;
   AIO_8302.VALUE_COEF := 0.00392;
   AIO_8007.AIO_CODE := 16#8007;
   AIO_8007.___________0020_0 := false;
   AIO_8007.___________0010_2 := false;
   AIO_8007.RAW_MIN := -12000;
   AIO_8007.RAW_MAX := 13000;
   AIO_8007.RAW_NAME := 'Thermal Resistance - 3-wire (Pt200 climate - 3851)';
   AIO_8007.___________0030_1 := false;
   AIO_8007.___________0030_2 := false;
   AIO_8007.PARAM_TYPE := 16#07;
   AIO_8007.PARAM_RANGE := 16#07;
   AIO_8007.PARAM_COEF := 16#00;
   AIO_8007.VALUE_COEF := 0.003851;
   AIO_8207.AIO_CODE := 16#8207;
   AIO_8207.___________0020_0 := false;
   AIO_8207.___________0010_2 := false;
   AIO_8207.RAW_MIN := -12000;
   AIO_8207.RAW_MAX := 13000;
   AIO_8207.RAW_NAME := 'Thermal Resistance - 3-wire (Pt200 climate - 3902)';
   AIO_8207.___________0030_1 := false;
   AIO_8207.___________0030_2 := false;
   AIO_8207.PARAM_TYPE := 16#07;
   AIO_8207.PARAM_RANGE := 16#07;
   AIO_8207.PARAM_COEF := 16#02;
   AIO_8207.VALUE_COEF := 0.003902;
   AIO_8507.AIO_CODE := 16#8507;
   AIO_8507.___________0020_0 := false;
   AIO_8507.___________0010_2 := false;
   AIO_8507.RAW_MIN := -12000;
   AIO_8507.RAW_MAX := 13000;
   AIO_8507.RAW_NAME := 'Thermal Resistance - 3-wire (Pt200 climate - 391)';
   AIO_8507.___________0030_1 := false;
   AIO_8507.___________0030_2 := false;
   AIO_8507.PARAM_TYPE := 16#07;
   AIO_8507.PARAM_RANGE := 16#07;
   AIO_8507.PARAM_COEF := 16#05;
   AIO_8507.VALUE_COEF := 0.00391;
   AIO_8107.AIO_CODE := 16#8107;
   AIO_8107.___________0020_0 := false;
   AIO_8107.___________0010_2 := false;
   AIO_8107.RAW_MIN := -12000;
   AIO_8107.RAW_MAX := 13000;
   AIO_8107.RAW_NAME := 'Thermal Resistance - 3-wire (Pt200 climate - 3916)';
   AIO_8107.___________0030_1 := false;
   AIO_8107.___________0030_2 := false;
   AIO_8107.PARAM_TYPE := 16#07;
   AIO_8107.PARAM_RANGE := 16#07;
   AIO_8107.PARAM_COEF := 16#01;
   AIO_8107.VALUE_COEF := 0.003916;
   AIO_8307.AIO_CODE := 16#8307;
   AIO_8307.___________0020_0 := false;
   AIO_8307.___________0010_2 := false;
   AIO_8307.RAW_MIN := -12000;
   AIO_8307.RAW_MAX := 13000;
   AIO_8307.RAW_NAME := 'Thermal Resistance - 3-wire (Pt200 climate - 392)';
   AIO_8307.___________0030_1 := false;
   AIO_8307.___________0030_2 := false;
   AIO_8307.PARAM_TYPE := 16#07;
   AIO_8307.PARAM_RANGE := 16#07;
   AIO_8307.PARAM_COEF := 16#03;
   AIO_8307.VALUE_COEF := 0.00392;
   AIO_800B.AIO_CODE := 16#800B;
   AIO_800B.___________0020_0 := false;
   AIO_800B.___________0010_2 := false;
   AIO_800B.RAW_MIN := -2000;
   AIO_800B.RAW_MAX := 8500;
   AIO_800B.RAW_NAME := 'Thermal Resistance - 3-wire (Pt200 standard - 3851)';
   AIO_800B.___________0030_1 := false;
   AIO_800B.___________0030_2 := false;
   AIO_800B.PARAM_TYPE := 16#07;
   AIO_800B.PARAM_RANGE := 16#0B;
   AIO_800B.PARAM_COEF := 16#00;
   AIO_800B.VALUE_COEF := 0.003851;
   AIO_820B.AIO_CODE := 16#820B;
   AIO_820B.___________0020_0 := false;
   AIO_820B.___________0010_2 := false;
   AIO_820B.RAW_MIN := -2000;
   AIO_820B.RAW_MAX := 8500;
   AIO_820B.RAW_NAME := 'Thermal Resistance - 3-wire (Pt200 standard - 3902)';
   AIO_820B.___________0030_1 := false;
   AIO_820B.___________0030_2 := false;
   AIO_820B.PARAM_TYPE := 16#07;
   AIO_820B.PARAM_RANGE := 16#0B;
   AIO_820B.PARAM_COEF := 16#02;
   AIO_820B.VALUE_COEF := 0.003902;
   AIO_850B.AIO_CODE := 16#850B;
   AIO_850B.___________0020_0 := false;
   AIO_850B.___________0010_2 := false;
   AIO_850B.RAW_MIN := -2000;
   AIO_850B.RAW_MAX := 8500;
   AIO_850B.RAW_NAME := 'Thermal Resistance - 3-wire (Pt200 standard - 391)';
   AIO_850B.___________0030_1 := false;
   AIO_850B.___________0030_2 := false;
   AIO_850B.PARAM_TYPE := 16#07;
   AIO_850B.PARAM_RANGE := 16#0B;
   AIO_850B.PARAM_COEF := 16#05;
   AIO_850B.VALUE_COEF := 0.00391;
   AIO_810B.AIO_CODE := 16#810B;
   AIO_810B.___________0020_0 := false;
   AIO_810B.___________0010_2 := false;
   AIO_810B.RAW_MIN := -2000;
   AIO_810B.RAW_MAX := 8500;
   AIO_810B.RAW_NAME := 'Thermal Resistance - 3-wire (Pt200 standard - 3916)';
   AIO_810B.___________0030_1 := false;
   AIO_810B.___________0030_2 := false;
   AIO_810B.PARAM_TYPE := 16#07;
   AIO_810B.PARAM_RANGE := 16#0B;
   AIO_810B.PARAM_COEF := 16#01;
   AIO_810B.VALUE_COEF := 0.003916;
   AIO_830B.AIO_CODE := 16#830B;
   AIO_830B.___________0020_0 := false;
   AIO_830B.___________0010_2 := false;
   AIO_830B.RAW_MIN := -2000;
   AIO_830B.RAW_MAX := 8500;
   AIO_830B.RAW_NAME := 'Thermal Resistance - 3-wire (Pt200 standard - 392)';
   AIO_830B.___________0030_1 := false;
   AIO_830B.___________0030_2 := false;
   AIO_830B.PARAM_TYPE := 16#07;
   AIO_830B.PARAM_RANGE := 16#0B;
   AIO_830B.PARAM_COEF := 16#03;
   AIO_830B.VALUE_COEF := 0.00392;
   AIO_8008.AIO_CODE := 16#8008;
   AIO_8008.___________0020_0 := false;
   AIO_8008.___________0010_2 := false;
   AIO_8008.RAW_MIN := -12000;
   AIO_8008.RAW_MAX := 13000;
   AIO_8008.RAW_NAME := 'Thermal Resistance - 3-wire (Pt500 climate - 3851)';
   AIO_8008.___________0030_1 := false;
   AIO_8008.___________0030_2 := false;
   AIO_8008.PARAM_TYPE := 16#07;
   AIO_8008.PARAM_RANGE := 16#08;
   AIO_8008.PARAM_COEF := 16#00;
   AIO_8008.VALUE_COEF := 0.003851;
   AIO_8208.AIO_CODE := 16#8208;
   AIO_8208.___________0020_0 := false;
   AIO_8208.___________0010_2 := false;
   AIO_8208.RAW_MIN := -12000;
   AIO_8208.RAW_MAX := 13000;
   AIO_8208.RAW_NAME := 'Thermal Resistance - 3-wire (Pt500 climate - 3902)';
   AIO_8208.___________0030_1 := false;
   AIO_8208.___________0030_2 := false;
   AIO_8208.PARAM_TYPE := 16#07;
   AIO_8208.PARAM_RANGE := 16#08;
   AIO_8208.PARAM_COEF := 16#02;
   AIO_8208.VALUE_COEF := 0.003902;
   AIO_8508.AIO_CODE := 16#8508;
   AIO_8508.___________0020_0 := false;
   AIO_8508.___________0010_2 := false;
   AIO_8508.RAW_MIN := -12000;
   AIO_8508.RAW_MAX := 13000;
   AIO_8508.RAW_NAME := 'Thermal Resistance - 3-wire (Pt500 climate - 391)';
   AIO_8508.___________0030_1 := false;
   AIO_8508.___________0030_2 := false;
   AIO_8508.PARAM_TYPE := 16#07;
   AIO_8508.PARAM_RANGE := 16#08;
   AIO_8508.PARAM_COEF := 16#05;
   AIO_8508.VALUE_COEF := 0.00391;
   AIO_8108.AIO_CODE := 16#8108;
   AIO_8108.___________0020_0 := false;
   AIO_8108.___________0010_2 := false;
   AIO_8108.RAW_MIN := -12000;
   AIO_8108.RAW_MAX := 13000;
   AIO_8108.RAW_NAME := 'Thermal Resistance - 3-wire (Pt500 climate - 3916)';
   AIO_8108.___________0030_1 := false;
   AIO_8108.___________0030_2 := false;
   AIO_8108.PARAM_TYPE := 16#07;
   AIO_8108.PARAM_RANGE := 16#08;
   AIO_8108.PARAM_COEF := 16#01;
   AIO_8108.VALUE_COEF := 0.003916;
   AIO_8308.AIO_CODE := 16#8308;
   AIO_8308.___________0020_0 := false;
   AIO_8308.___________0010_2 := false;
   AIO_8308.RAW_MIN := -12000;
   AIO_8308.RAW_MAX := 13000;
   AIO_8308.RAW_NAME := 'Thermal Resistance - 3-wire (Pt500 climate - 392)';
   AIO_8308.___________0030_1 := false;
   AIO_8308.___________0030_2 := false;
   AIO_8308.PARAM_TYPE := 16#07;
   AIO_8308.PARAM_RANGE := 16#08;
   AIO_8308.PARAM_COEF := 16#03;
   AIO_8308.VALUE_COEF := 0.00392;
   AIO_8004.AIO_CODE := 16#8004;
   AIO_8004.___________0020_0 := false;
   AIO_8004.___________0010_2 := false;
   AIO_8004.RAW_MIN := -2000;
   AIO_8004.RAW_MAX := 8500;
   AIO_8004.RAW_NAME := 'Thermal Resistance - 3-wire (Pt500 standard - 3851)';
   AIO_8004.___________0030_1 := false;
   AIO_8004.___________0030_2 := false;
   AIO_8004.PARAM_TYPE := 16#07;
   AIO_8004.PARAM_RANGE := 16#04;
   AIO_8004.PARAM_COEF := 16#00;
   AIO_8004.VALUE_COEF := 0.003851;
   AIO_8204.AIO_CODE := 16#8204;
   AIO_8204.___________0020_0 := false;
   AIO_8204.___________0010_2 := false;
   AIO_8204.RAW_MIN := -2000;
   AIO_8204.RAW_MAX := 8500;
   AIO_8204.RAW_NAME := 'Thermal Resistance - 3-wire (Pt500 standard - 3902)';
   AIO_8204.___________0030_1 := false;
   AIO_8204.___________0030_2 := false;
   AIO_8204.PARAM_TYPE := 16#07;
   AIO_8204.PARAM_RANGE := 16#04;
   AIO_8204.PARAM_COEF := 16#02;
   AIO_8204.VALUE_COEF := 0.003902;
   AIO_8504.AIO_CODE := 16#8504;
   AIO_8504.___________0020_0 := false;
   AIO_8504.___________0010_2 := false;
   AIO_8504.RAW_MIN := -2000;
   AIO_8504.RAW_MAX := 8500;
   AIO_8504.RAW_NAME := 'Thermal Resistance - 3-wire (Pt500 standard - 391)';
   AIO_8504.___________0030_1 := false;
   AIO_8504.___________0030_2 := false;
   AIO_8504.PARAM_TYPE := 16#07;
   AIO_8504.PARAM_RANGE := 16#04;
   AIO_8504.PARAM_COEF := 16#05;
   AIO_8504.VALUE_COEF := 0.00391;
   AIO_8104.AIO_CODE := 16#8104;
   AIO_8104.___________0020_0 := false;
   AIO_8104.___________0010_2 := false;
   AIO_8104.RAW_MIN := -2000;
   AIO_8104.RAW_MAX := 8500;
   AIO_8104.RAW_NAME := 'Thermal Resistance - 3-wire (Pt500 standard - 3916)';
   AIO_8104.___________0030_1 := false;
   AIO_8104.___________0030_2 := false;
   AIO_8104.PARAM_TYPE := 16#07;
   AIO_8104.PARAM_RANGE := 16#04;
   AIO_8104.PARAM_COEF := 16#01;
   AIO_8104.VALUE_COEF := 0.003916;
   AIO_8304.AIO_CODE := 16#8304;
   AIO_8304.___________0020_0 := false;
   AIO_8304.___________0010_2 := false;
   AIO_8304.RAW_MIN := -2000;
   AIO_8304.RAW_MAX := 8500;
   AIO_8304.RAW_NAME := 'Thermal Resistance - 3-wire (Pt500 standard - 392)';
   AIO_8304.___________0030_1 := false;
   AIO_8304.___________0030_2 := false;
   AIO_8304.PARAM_TYPE := 16#07;
   AIO_8304.PARAM_RANGE := 16#04;
   AIO_8304.PARAM_COEF := 16#03;
   AIO_8304.VALUE_COEF := 0.00392;
   AIO_8009.AIO_CODE := 16#8009;
   AIO_8009.___________0020_0 := false;
   AIO_8009.___________0010_2 := false;
   AIO_8009.RAW_MIN := -12000;
   AIO_8009.RAW_MAX := 13000;
   AIO_8009.RAW_NAME := 'Thermal Resistance - 3-wire (Pt1000 climate - 3851)';
   AIO_8009.___________0030_1 := false;
   AIO_8009.___________0030_2 := false;
   AIO_8009.PARAM_TYPE := 16#07;
   AIO_8009.PARAM_RANGE := 16#09;
   AIO_8009.PARAM_COEF := 16#00;
   AIO_8009.VALUE_COEF := 0.003851;
   AIO_8209.AIO_CODE := 16#8209;
   AIO_8209.___________0020_0 := false;
   AIO_8209.___________0010_2 := false;
   AIO_8209.RAW_MIN := -12000;
   AIO_8209.RAW_MAX := 13000;
   AIO_8209.RAW_NAME := 'Thermal Resistance - 3-wire (Pt1000 climate - 3902)';
   AIO_8209.___________0030_1 := false;
   AIO_8209.___________0030_2 := false;
   AIO_8209.PARAM_TYPE := 16#07;
   AIO_8209.PARAM_RANGE := 16#09;
   AIO_8209.PARAM_COEF := 16#02;
   AIO_8209.VALUE_COEF := 0.003902;
   AIO_8509.AIO_CODE := 16#8509;
   AIO_8509.___________0020_0 := false;
   AIO_8509.___________0010_2 := false;
   AIO_8509.RAW_MIN := -12000;
   AIO_8509.RAW_MAX := 13000;
   AIO_8509.RAW_NAME := 'Thermal Resistance - 3-wire (Pt1000 climate - 391)';
   AIO_8509.___________0030_1 := false;
   AIO_8509.___________0030_2 := false;
   AIO_8509.PARAM_TYPE := 16#07;
   AIO_8509.PARAM_RANGE := 16#09;
   AIO_8509.PARAM_COEF := 16#05;
   AIO_8509.VALUE_COEF := 0.00391;
   AIO_8109.AIO_CODE := 16#8109;
   AIO_8109.___________0020_0 := false;
   AIO_8109.___________0010_2 := false;
   AIO_8109.RAW_MIN := -12000;
   AIO_8109.RAW_MAX := 13000;
   AIO_8109.RAW_NAME := 'Thermal Resistance - 3-wire (Pt1000 climate - 3916)';
   AIO_8109.___________0030_1 := false;
   AIO_8109.___________0030_2 := false;
   AIO_8109.PARAM_TYPE := 16#07;
   AIO_8109.PARAM_RANGE := 16#09;
   AIO_8109.PARAM_COEF := 16#01;
   AIO_8109.VALUE_COEF := 0.003916;
   AIO_8309.AIO_CODE := 16#8309;
   AIO_8309.___________0020_0 := false;
   AIO_8309.___________0010_2 := false;
   AIO_8309.RAW_MIN := -12000;
   AIO_8309.RAW_MAX := 13000;
   AIO_8309.RAW_NAME := 'Thermal Resistance - 3-wire (Pt1000 climate - 392)';
   AIO_8309.___________0030_1 := false;
   AIO_8309.___________0030_2 := false;
   AIO_8309.PARAM_TYPE := 16#07;
   AIO_8309.PARAM_RANGE := 16#09;
   AIO_8309.PARAM_COEF := 16#03;
   AIO_8309.VALUE_COEF := 0.00392;
   AIO_8005.AIO_CODE := 16#8005;
   AIO_8005.___________0020_0 := false;
   AIO_8005.___________0010_2 := false;
   AIO_8005.RAW_MIN := -2000;
   AIO_8005.RAW_MAX := 8500;
   AIO_8005.RAW_NAME := 'Thermal Resistance - 3-wire (Pt1000 standard - 3851)';
   AIO_8005.___________0030_1 := false;
   AIO_8005.___________0030_2 := false;
   AIO_8005.PARAM_TYPE := 16#07;
   AIO_8005.PARAM_RANGE := 16#05;
   AIO_8005.PARAM_COEF := 16#00;
   AIO_8005.VALUE_COEF := 0.003851;
   AIO_8205.AIO_CODE := 16#8205;
   AIO_8205.___________0020_0 := false;
   AIO_8205.___________0010_2 := false;
   AIO_8205.RAW_MIN := -2000;
   AIO_8205.RAW_MAX := 8500;
   AIO_8205.RAW_NAME := 'Thermal Resistance - 3-wire (Pt1000 standard - 3902)';
   AIO_8205.___________0030_1 := false;
   AIO_8205.___________0030_2 := false;
   AIO_8205.PARAM_TYPE := 16#07;
   AIO_8205.PARAM_RANGE := 16#05;
   AIO_8205.PARAM_COEF := 16#02;
   AIO_8205.VALUE_COEF := 0.003902;
   AIO_8505.AIO_CODE := 16#8505;
   AIO_8505.___________0020_0 := false;
   AIO_8505.___________0010_2 := false;
   AIO_8505.RAW_MIN := -2000;
   AIO_8505.RAW_MAX := 8500;
   AIO_8505.RAW_NAME := 'Thermal Resistance - 3-wire (Pt1000 standard - 391)';
   AIO_8505.___________0030_1 := false;
   AIO_8505.___________0030_2 := false;
   AIO_8505.PARAM_TYPE := 16#07;
   AIO_8505.PARAM_RANGE := 16#05;
   AIO_8505.PARAM_COEF := 16#05;
   AIO_8505.VALUE_COEF := 0.00391;
   AIO_8105.AIO_CODE := 16#8105;
   AIO_8105.___________0020_0 := false;
   AIO_8105.___________0010_2 := false;
   AIO_8105.RAW_MIN := -2000;
   AIO_8105.RAW_MAX := 8500;
   AIO_8105.RAW_NAME := 'Thermal Resistance - 3-wire (Pt1000 standard - 3916)';
   AIO_8105.___________0030_1 := false;
   AIO_8105.___________0030_2 := false;
   AIO_8105.PARAM_TYPE := 16#07;
   AIO_8105.PARAM_RANGE := 16#05;
   AIO_8105.PARAM_COEF := 16#01;
   AIO_8105.VALUE_COEF := 0.003916;
   AIO_8305.AIO_CODE := 16#8305;
   AIO_8305.___________0020_0 := false;
   AIO_8305.___________0010_2 := false;
   AIO_8305.RAW_MIN := -2000;
   AIO_8305.RAW_MAX := 8500;
   AIO_8305.RAW_NAME := 'Thermal Resistance - 3-wire (Pt1000 standard - 392)';
   AIO_8305.___________0030_1 := false;
   AIO_8305.___________0030_2 := false;
   AIO_8305.PARAM_TYPE := 16#07;
   AIO_8305.PARAM_RANGE := 16#05;
   AIO_8305.PARAM_COEF := 16#03;
   AIO_8305.VALUE_COEF := 0.00392;
   AIO_A000.AIO_CODE := 16#A000;
   AIO_A000.___________0020_0 := false;
   AIO_A000.___________0010_2 := false;
   AIO_A000.RAW_MIN := 2500;
   AIO_A000.RAW_MAX := 18200;
   AIO_A000.RAW_NAME := 'Thermocouple (Type B)';
   AIO_A000.___________0030_1 := false;
   AIO_A000.___________0030_2 := false;
   AIO_A000.PARAM_TYPE := 16#0A;
   AIO_A000.PARAM_RANGE := 16#00;
   AIO_A000.PARAM_COEF := 16#00;
   AIO_A00A.AIO_CODE := 16#A00A;
   AIO_A00A.___________0020_0 := false;
   AIO_A00A.___________0010_2 := false;
   AIO_A00A.RAW_MIN := 0;
   AIO_A00A.RAW_MAX := 23000;
   AIO_A00A.RAW_NAME := 'Thermocouple (Type C)';
   AIO_A00A.___________0030_1 := false;
   AIO_A00A.___________0030_2 := false;
   AIO_A00A.PARAM_TYPE := 16#0A;
   AIO_A00A.PARAM_RANGE := 16#0A;
   AIO_A00A.PARAM_COEF := 16#00;
   AIO_A002.AIO_CODE := 16#A002;
   AIO_A002.___________0020_0 := false;
   AIO_A002.___________0010_2 := false;
   AIO_A002.RAW_MIN := -2700;
   AIO_A002.RAW_MAX := 12000;
   AIO_A002.RAW_NAME := 'Thermocouple (Type E)';
   AIO_A002.___________0030_1 := false;
   AIO_A002.___________0030_2 := false;
   AIO_A002.PARAM_TYPE := 16#0A;
   AIO_A002.PARAM_RANGE := 16#02;
   AIO_A002.PARAM_COEF := 16#00;
   AIO_A005.AIO_CODE := 16#A005;
   AIO_A005.___________0020_0 := false;
   AIO_A005.___________0010_2 := false;
   AIO_A005.RAW_MIN := -2100;
   AIO_A005.RAW_MAX := 12000;
   AIO_A005.RAW_NAME := 'Thermocouple (Type J)';
   AIO_A005.___________0030_1 := false;
   AIO_A005.___________0030_2 := false;
   AIO_A005.PARAM_TYPE := 16#0A;
   AIO_A005.PARAM_RANGE := 16#05;
   AIO_A005.PARAM_COEF := 16#00;
   AIO_A008.AIO_CODE := 16#A008;
   AIO_A008.___________0020_0 := false;
   AIO_A008.___________0010_2 := false;
   AIO_A008.RAW_MIN := -2700;
   AIO_A008.RAW_MAX := 13720;
   AIO_A008.RAW_NAME := 'Thermocouple (Type K)';
   AIO_A008.___________0030_1 := false;
   AIO_A008.___________0030_2 := false;
   AIO_A008.PARAM_TYPE := 16#0A;
   AIO_A008.PARAM_RANGE := 16#08;
   AIO_A008.PARAM_COEF := 16#00;
   AIO_A001.AIO_CODE := 16#A001;
   AIO_A001.___________0020_0 := false;
   AIO_A001.___________0010_2 := false;
   AIO_A001.RAW_MIN := -2700;
   AIO_A001.RAW_MAX := 13000;
   AIO_A001.RAW_NAME := 'Thermocouple (Type N)';
   AIO_A001.___________0030_1 := false;
   AIO_A001.___________0030_2 := false;
   AIO_A001.PARAM_TYPE := 16#0A;
   AIO_A001.PARAM_RANGE := 16#01;
   AIO_A001.PARAM_COEF := 16#00;
   AIO_A003.AIO_CODE := 16#A003;
   AIO_A003.___________0020_0 := false;
   AIO_A003.___________0010_2 := false;
   AIO_A003.RAW_MIN := -500;
   AIO_A003.RAW_MAX := 17690;
   AIO_A003.RAW_NAME := 'Thermocouple (Type R)';
   AIO_A003.___________0030_1 := false;
   AIO_A003.___________0030_2 := false;
   AIO_A003.PARAM_TYPE := 16#0A;
   AIO_A003.PARAM_RANGE := 16#03;
   AIO_A003.PARAM_COEF := 16#00;
   AIO_A004.AIO_CODE := 16#A004;
   AIO_A004.___________0020_0 := false;
   AIO_A004.___________0010_2 := false;
   AIO_A004.RAW_MIN := -500;
   AIO_A004.RAW_MAX := 17690;
   AIO_A004.RAW_NAME := 'Thermocouple (Type S)';
   AIO_A004.___________0030_1 := false;
   AIO_A004.___________0030_2 := false;
   AIO_A004.PARAM_TYPE := 16#0A;
   AIO_A004.PARAM_RANGE := 16#04;
   AIO_A004.PARAM_COEF := 16#00;
   AIO_A007.AIO_CODE := 16#A007;
   AIO_A007.___________0020_0 := false;
   AIO_A007.___________0010_2 := false;
   AIO_A007.RAW_MIN := -2700;
   AIO_A007.RAW_MAX := 4000;
   AIO_A007.RAW_NAME := 'Thermocouple (Type T)';
   AIO_A007.___________0030_1 := false;
   AIO_A007.___________0030_2 := false;
   AIO_A007.PARAM_TYPE := 16#0A;
   AIO_A007.PARAM_RANGE := 16#07;
   AIO_A007.PARAM_COEF := 16#00;
   AIO_A00B.AIO_CODE := 16#A00B;
   AIO_A00B.___________0020_0 := false;
   AIO_A00B.___________0010_2 := false;
   AIO_A00B.RAW_MIN := -2000;
   AIO_A00B.RAW_MAX := 8000;
   AIO_A00B.RAW_NAME := 'Thermocouple (Type TXK/XCL)';
   AIO_A00B.___________0030_1 := false;
   AIO_A00B.___________0030_2 := false;
   AIO_A00B.PARAM_TYPE := 16#0A;
   AIO_A00B.PARAM_RANGE := 16#0B;
   AIO_A00B.PARAM_COEF := 16#00;
END_DATA_BLOCK
